PROGRAM MAIN
VAR
	CallButtons:ARRAY[1..numFloor]OF BOOL;
	Floor:ARRAY[1..numFloor]OF ST_Floor;
	Elevator:FB_Motor;
	PrgState:UINT;
	current: INT;
	requested: INT;
	i: INT;
	Rise:ARRAY[1..numFloor] OF R_TRIG;
END_VAR
VAR CONSTANT
	numFloor:UINT:=6;
END_VAR

CASE	PrgState	OF
	0://stopped
		IF	current<requested	THEN
			PrgState:=20;//change state to moveing up
			Elevator.MoveUP();
		ELSIF current>requested	THEN
			PrgState:=30;//change state to moveing down
			Elevator.MoveDown();
		ELSE
			PrgState:=10;//poll for inputs
		END_IF
	10://poll input
		FOR	i:=1	TO	numFloor	DO
			IF	CallButtons[i]	THEN
				requested:=i;
				EXIT;
			END_IF
		END_FOR
		PrgState:=0;
	20://moveing up
		FOR i:=1	TO	numFloor	DO
			Rise[i](CLK:= Floor[i].Low,);
			IF	Rise[i].Q	THEN
				current:=current+1;
				IF	current=requested	THEN
					PrgState:=40;
				ELSE
					CONTINUE;
				END_IF
			ELSE
				CONTINUE;
			END_IF
		END_FOR
	30://moving down
		FOR i:=1	TO	numFloor	DO
			Rise[i](CLK:= Floor[i].High,);
			IF	Rise[i].Q	THEN
				current:=current-1;
				IF	current=requested	THEN
					PrgState:=40;
				ELSE
					CONTINUE;
				END_IF
			ELSE
				CONTINUE;
			END_IF
		END_FOR
	40://slowdown
		Elevator.SlowDown();
		FOR i:=1	TO	numFloor	DO
			IF	Floor[i].Mid	THEN
				Elevator.Stop();
				EXIT;
			END_IF
		END_FOR
		IF	elevator.IsStopped()	THEN
			PrgState:=0;
		END_IF
END_CASE

END_PROGRAM

(* stored: Version 1.1.0.1, ProductVersion 3.1.4024.11
   POU MAIN: Id {102166ba-9c0f-48e5-baec-6e460cabbb86}, SpecialFunc None *)
